{attribute 'no_explicit_call' := 'do not call this POU directly'}
{attribute 'conditionalshow_all_locals'}
FUNCTION_BLOCK INTERNAL FINAL FB_RpcConfig IMPLEMENTS I_RpcDynamicConfigAmsNetId, I_RpcDynamicConfigAmsPort, I_RpcDynamicConfigSymbolPath, I_RpcDynamicConfigBuild
VAR_INPUT
END_VAR
VAR_OUTPUT
END_VAR
VAR	
	sAmsNetIdLocalField		: T_AmsNetId;
	nAmsPortLocalField		: T_AmsPort;
	sInstancePathLocalField	: STRING;
	sSymbolLocalField		: STRING;
	pFbRpcBase				: POINTER TO FB_RpcBase;
END_VAR

METHOD Build : HRESULT
IF pFbRpcBase = NULL THEN
	Build := E_HRESULTAdsErr.INVALIDINTERFACE;
	RETURN;
END_IF
Build := pFbRpcBase^.ConfigDoneCallBack(sAmsNetId:= sAmsNetIdLocalField, nAmsPort:= nAmsPortLocalField, sInstancePath:= sInstancePathLocalField, sSymbol:= sSymbolLocalField);
END_METHOD

METHOD INTERNAL SetCallback
VAR_INPUT
	pFbRpcBase : POINTER TO FB_RpcBase;
END_VAR
THIS^.pFbRpcBase := pFbRpcBase;
END_METHOD

METHOD WithAmsNetId : I_RpcDynamicConfigAmsPort
VAR_INPUT
	sAmsNetId	: Tc2_System.T_AmsNetID;
END_VAR
THIS^.sAmsNetIdLocalField := sAmsNetId;

WithAmsNetId := THIS^;
END_METHOD

METHOD WithAmsPort : I_RpcDynamicConfigSymbolPath
VAR_INPUT
	nAmsPort	: Tc2_System.T_AmsPort;
END_VAR
THIS^.nAmsPortLocalField := nAmsPort;

WithAmsPort := THIS^;
END_METHOD

METHOD WithSymbolPath : I_RpcDynamicConfigBuild
VAR_INPUT
	sInstancePath	: STRING;
	sSymbol	: STRING;
END_VAR
THIS^.sInstancePathLocalField := sInstancePath;
THIS^.sSymbolLocalField := sSymbol;

WithSymbolPath := THIS^;
END_METHOD

END_FUNCTION_BLOCK

(* stored: Version 1.1.0.1, ProductVersion 3.1.4024.12
   POU FB_RpcConfig: Id {0ece8654-785d-4f03-8887-a8736c00785e}, SpecialFunc None
   Folder ITFs: Id {bb2aed01-6a79-4ef6-b50d-acc2f5488200}
   Method Build: Id {b68bc296-e290-4099-b447-5264915e1e6a}
   Method SetCallback: Id {ea8a6ec3-f23f-411d-8f63-3d4035460924}
   Method WithAmsNetId: Id {b82ba08f-7e00-440a-8f8e-76f93109c9d8}
   Method WithAmsPort: Id {24232020-6a85-4d8d-9bce-84f9c8bbcda5}
   Method WithSymbolPath: Id {6d75d2e7-e55a-4750-9698-dde9afeecb9e} *)
